Universal Robots PolyScope program: RC_E7_PICK_720.urp

Program RC_E7_PICK_720 (createdIn=3.0.0 lastSavedIn=3.0.0 directory=/programs installation=default)
Robot Program (runOnlyOnce=true motionType=MoveJ speed=1.047198 acceleration=1.396263 useActiveTCP=false)
  'Program generated by RoboDK v4.1.0 for UR3e_HORNO on 05/09/2022 13:23:39'
  'Using nominal kinematics.'
  'Using Ref. Frame RC Traslado B: p[0.370000, -0.335000, 0.000000, 0.000000, 0.000000, 0.000000]'
  'Using TCP 0208-0001-0001-307-000-3 Horno: p[0.000000, 0.000000, 0.164750, 0.000000, 0.000000, 0.000000]'
  Script: set_tcp(p[0.000000, 0.000000, 0.164750, 0.000000, 0.000000, 0.000000])
  Script: movej([-0.630226, -2.201890, -0.581884, -1.909474, 1.548658, 0.946153],0.60000,0.12500,0,0.0000)
  Script: movej([-0.700570, -2.446385, -0.858486, -1.402697, 1.567730, 0.875467],0.60000,0.12500,0,0.0000)
  'Attach to 0208-0001-0001-307-000-3 Horno'
  MoveL speed 80 mm/s, acceleration 80 mm/s^2 (useActiveTCP=true)
    Waypoint Waypoint_1: TCP in base x=639.759 y=-701.028 z=168.101 mm, rx=0.0091 ry=3.1387 rz=-0.0458 rad; joints [-36.109, -126.159, -33.339, -109.405, 88.732, 54.211] deg; flange x=639.361 y=-696.224 z=332.78 mm, rx=0.0091 ry=3.1387 rz=-0.0458 rad
